// TIA Portal V20 export
// export: Created 2026-07-16T12:58:50.6487407Z, ExportSetting WithDefaults, DisplayName Totally Integrated Automation Portal, DisplayVersion V20 Update 5, DisplayName TIA Portal Openness, DisplayVersion V20 Update 4, DisplayName TIA Portal Version Control Interface, DisplayVersion V20 Update 5, DisplayName SINAMICS Startdrive Advanced, DisplayVersion V20, DisplayName SINAMICS DCC, DisplayVersion V20, DisplayName SINAMICS Startdrive G130, G150, S120, S150, SINAMICS MV, G220, S200, S210, DisplayVersion V20, DisplayName SINAMICS Startdrive G110M, G120, G120C, G120D, G120P, G115D, DisplayVersion V20, DisplayName STEP 7 Professional, DisplayVersion V20 Update 5, DisplayName STEP 7 Safety, DisplayVersion V20 Update 2, DisplayName WinCC Basic/Comfort/Advanced, DisplayVersion V20 Update 5, DisplayName WinCC Unified, DisplayVersion V20 Update 5
DATA_BLOCK "iDB_ShredderSequencer"   // DB11
VERSION : 0.1
// stored: AutoNumber true, DBAccessibleFromOPCUA true, InstanceOfName FB_ShredderSequencer, InstanceOfType FB
"FB_ShredderSequencer"
   // VAR RETAIN
   //    IO { S7_SetPoint := 'True'} : "UDT_ShredderSequencerIO";
   // END_VAR
   // VAR
   //    StopCmd : Bool;
   //    ReversalWindowTimeMS : DInt;
   //    PreStartSounderTimeMS : DInt;
   //    DischargeConveyorTimeoutMS : DInt;
   //    ShredderReverseRunTimeMS : DInt;
   //    InfeedRestartDelayMS : DInt;
   //    InfeedToUpstreamEnableDelayMS : DInt;
   //    OvercurrentSpinUpAllowanceMS : DInt;
   //    OvercurrentMediumDelayMS : DInt;
   //    OvercurrentHighDelayMS : DInt;
   //    ReversalRetryPauseTimeMS : DInt;
   //    ReversalWindowTimer { S7_SetPoint := 'True'} : TON_TIME;
   //    ReversalStepEdge : Bool;
   //    ReversalStepEdgeMem : Bool;
   //    ReversalCount : Int;
   //    PreStartTimer { S7_SetPoint := 'True'} : TON_TIME;
   //    DischargeStartTimer { S7_SetPoint := 'True'} : TON_TIME;
   //    ReverseRunTimer { S7_SetPoint := 'True'} : TON_TIME;
   //    InfeedRestartTimer { S7_SetPoint := 'True'} : TON_TIME;
   //    UpstreamEnableTimer { S7_SetPoint := 'True'} : TON_TIME;
   //    InfeedRunning : Bool;
   //    SpinUpTimer { S7_SetPoint := 'True'} : TON_TIME;
   //    OvercurrentMediumTimer { S7_SetPoint := 'True'} : TON_TIME;
   //    OvercurrentHighTimer { S7_SetPoint := 'True'} : TON_TIME;
   //    OvercurrentTripped : Bool;
   //    OvercurrentAbortPauseTimer { S7_SetPoint := 'True'} : TON_TIME;
   // END_VAR
BEGIN
END_DATA_BLOCK
